// TIA Portal V19 export
DATA_BLOCK "RINSE-1_CLEANING"   // DB7
// stored: InstanceOfName TIMING_BLOCK, InstanceOfType FB
"TIMING_BLOCK"
   // VAR_INPUT
   //    "SET TIME" : Int;
   //    RESET : Bool;
   //    INPUT : Bool;
   // END_VAR
   // VAR_OUTPUT
   //    "PRESENT VALUE OF TIME" : Int;
   //    DONE : Bool;
   // END_VAR
   // VAR
   //    "TIMER 1" { S7_SetPoint := 'True'} : IEC_TIMER;
   // END_VAR
   // VAR RETAIN
   //    "COUNTER1 1" { S7_SetPoint := 'True'} : IEC_COUNTER;
   // END_VAR
BEGIN
END_DATA_BLOCK
